(* IEC 61131-3 sources: F100R_S278_Temperville/MyController.device.xml.v3^/Plc Logic.plclogic.xml.v3^/Application.application.xml.v3^/01_Inicialização, 3 files *)

(* ---- A_Inicializacao.prg.st ---- *)
PROGRAM A_Inicializacao
VAR
	///passo para logica de inicialização do sistema
	PassoInit: INT := 0;
	ContDrive: INT := 0;
	TonInicilizacaoSistema: TON;
	xTonInicilizacaoSistemaIn: BOOL;
	xTonInicilizacaoSistemaQ: BOOL;
	TonLeituraErroInicial: TON;
	xTonLeituraErroInicialIn: BOOL;
	xTonLeituraErroInicialQ: BOOL;
	tDelayIniSystem: TON;
	tDelayIniSystemIn: BOOL;
	tDelayIniSystemQ: BOOL;
	///atraso entre os passos 0 e 1
	AtrasoPasso01: TON;
	/// tempo limite para verificar se os drives foram habilitados
	AtrasoLeituraStatus: TON;
	/// tempo de reset
	AtrasoRstErro: TON;
	delayResetaNo: TON;
	AtrasoEstabilizaRede: TON;
	/// Ativa leitura dos drives
	xAtivaLeituraErro: BOOL;
	iContadorReset: INT;
	xCanOpenOk: BOOL;
	///Flag indicativo para falha na rede CanOpen ou CanMotion
	xCanOpenFh: BOOL;
	/// Bit para habilitar drives do sistema
	xHabilitaDrives: BOOL;
	/// bit para resetar alarmes
	xRstAlarmes: BOOL;
	///------------------------------------------------------------------------//
	///Mesa Entrada
	McResetMesaEntrada: GIPLC.MC_Reset;
	McPowerMesaEntrada: GIPLC.MC_Power;
	McReadStatusMesaEntrada: GIPLC.MC_ReadStatus;
	McReadErrorMesaEntrada: GIPLC.MC_ReadAxisError;
	///Mesa Forno
	McResetMesaForno: GIPLC.MC_Reset;
	McPowerMesaForno: GIPLC.MC_Power;
	McReadStatusMesaForno: GIPLC.MC_ReadStatus;
	McReadErrorMesaForno: GIPLC.MC_ReadAxisError;
	///Mesa Resfriamento
	McResetMesaResfriador: GIPLC.MC_Reset;
	McPowerMesaResfriador: GIPLC.MC_Power;
	McReadStatusMesaResfriado: GIPLC.MC_ReadStatus;
	McReadErrorMesaResfriador: GIPLC.MC_ReadAxisError;
	///Mesa Saída
	McResetMesaSaida: GIPLC.MC_Reset;
	McPowerMesaSaida: GIPLC.MC_Power;
	McReadStatusMesaSaida: GIPLC.MC_ReadStatus;
	McReadErrorMesaSaida: GIPLC.MC_ReadAxisError;
	///Ductos Inferior 01
	McResetDutosResfriadorInf01: GIPLC.MC_Reset;
	McPowerDutosResfriadorInf01: GIPLC.MC_Power;
	McReadDutosResfriadorInf01: GIPLC.MC_ReadStatus;
	McReadErrorDutosResfriadorInf01: GIPLC.MC_ReadAxisError;
	///Ductos Superior 01
	McResetDutosResfriadorSup01: GIPLC.MC_Reset;
	McPowerDutosResfriadorSup01: GIPLC.MC_Power;
	McReadDutosResfriadorSup01: GIPLC.MC_ReadStatus;
	McReadErrorDutosResfriadorSup01: GIPLC.MC_ReadAxisError;
	///Ductos Inferior 02
	McResetDutosResfriadorInf02: GIPLC.MC_Reset;
	McPowerDutosResfriadorInf02: GIPLC.MC_Power;
	McReadDutosResfriadorInf02: GIPLC.MC_ReadStatus;
	McReadErrorDutosResfriadorInf02: GIPLC.MC_ReadAxisError;
	///Ductos Superior 02
	McResetDutosResfriadorSup02: GIPLC.MC_Reset;
	McPowerDutosResfriadorSup02: GIPLC.MC_Power;
	McReadDutosResfriadorSup02: GIPLC.MC_ReadStatus;
	McReadErrorDutosResfriadorSup02: GIPLC.MC_ReadAxisError;
	///Guilhotina01
	McResetGuilhotina01: GIPLC.MC_Reset;
	McPowerGuilhotina01: GIPLC.MC_Power;
	McReadStatusGuilhotina01: GIPLC.MC_ReadStatus;
	McReadErrorGuilhotina01: GIPLC.MC_ReadAxisError;
	///Guilhotina02
	McResetGuilhotina02: GIPLC.MC_Reset;
	McPowerGuilhotina02: GIPLC.MC_Power;
	McReadStatusGuilhotina02: GIPLC.MC_ReadStatus;
	McReadErrorGuilhotina02: GIPLC.MC_ReadAxisError;
	/// Motor Limpeza Resfriador 02
	McResetLimpResfriadorSup02: GIPLC.MC_Reset;
	McPowerLimpResfriadorSup02: GIPLC.MC_Power;
	McReadStatusLimpResfriadorSup02: GIPLC.MC_ReadStatus;
	McReadErrorLimpResfriadorSup02: GIPLC.MC_ReadAxisError;
	/// Motor Abertura Caixa do Forno
	McResetCaixaForno: GIPLC.MC_Reset;
	McPowerCaixaForno: GIPLC.MC_Power;
	McReadStatusCaixaForno: GIPLC.MC_ReadStatus;
	McReadErrorCaixaForno: GIPLC.MC_ReadAxisError;
	///Ventilador01
	McResetVentilador01: GIPLC.MC_Reset;
	McPowerVentilador01: GIPLC.MC_Power;
	McReadStatusVentilador01: GIPLC.MC_ReadStatus;
	McReadErrorVentilador01: GIPLC.MC_ReadAxisError;
	PulsoRstVent01Auto: TP;
	///Ventilador02
	McResetVentilador02: GIPLC.MC_Reset;
	McPowerVentilador02: GIPLC.MC_Power;
	McReadStatusVentilador02: GIPLC.MC_ReadStatus;
	McReadErrorVentilador02: GIPLC.MC_ReadAxisError;
	PulsoRstVent02Auto: TP;
	///Ventilador03
	McResetVentilador03: GIPLC.MC_Reset;
	McPowerVentilador03: GIPLC.MC_Power;
	McReadStatusVentilador03: GIPLC.MC_ReadStatus;
	McReadErrorVentilador03: GIPLC.MC_ReadAxisError;
	PulsoRstVent03Auto: TP;
	///Ventilador03
	McResetVentilador04: GIPLC.MC_Reset;
	McPowerVentilador04: GIPLC.MC_Power;
	McReadStatusVentilador04: GIPLC.MC_ReadStatus;
	McReadErrorVentilador04: GIPLC.MC_ReadAxisError;
	PulsoRstVent04Auto: TP;
	///Ventilador Convecção
	McResetVentConvec: GIPLC.MC_Reset;
	McPowerVentConvec: GIPLC.MC_Power;
	McReadStatusVentConvec: GIPLC.MC_ReadStatus;
	McReadErrorVentConvec: GIPLC.MC_ReadAxisError;
	///-----------------------------------------------------------------------//
	xResetErroVent03: BOOL;
	///----------------------------------------------------------------------//
	xErroDeEixo: BOOL;
	ResetaRedeCanOpen: CIA405.NMT;
	iNdevice: USINT := 1;
	testemsl: BOOL;
	AuxResetRedeCanOpen: BOOL;
	xInicializacaoOk: BOOL;
	xErroEixo: ARRAY[1..14] OF BOOL;
	xEixoHabilitado: ARRAY[1..14] OF BOOL;
	xHabilitaDriveMe: BOOL;
	xHabilitaDriveMf: BOOL;
	xHabilitaDriveMr: BOOL;
	xHabilitaDriveMs: BOOL;
	xHabilitaDriveMdI01: BOOL;
	xHabilitaDriveMdS01: BOOL;
	xHabilitaDriveMdI02: BOOL;
	xHabilitaDriveMdS02: BOOL;
	xHabilitaDriveMg01: BOOL;
	xHabilitaDriveMg02: BOOL;
	xHabilitaDriveMv01: BOOL;
	xHabilitaDriveMv02: BOOL;
	xHabilitaDriveMv03: BOOL;
	xHabilitaDriveMv04: BOOL;
	xResetErroVentilador01: BOOL;
	xResetErroVentilador02: BOOL;
	xResetErroVentilador03: BOOL;
	xResetErroVentilador04: BOOL;
	xHabilitaDriveMvC: BOOL;
	xResetErroMe: BOOL;
	xResetErroMf: BOOL;
	xResetErroMr: BOOL;
	xResetErroMs: BOOL;
	xResetErroMdS02: BOOL;
	xResetErroMg02: BOOL;
	xResetErroV03: BOOL;
	xResetErroV04: BOOL;
END_VAR

iNumResistencias:=iNumeroResistencias/2;

(* ---- ComunicacaoOpc.prg.st ---- *)
PROGRAM ComunicacaoOpc
VAR
	xEnviaSuperClp: INT;
	xRecebeClpSuper: INT;
	ton01: ton;
	ton01In: BOOL;
END_VAR
VAR_OUTPUT
	ton01Q: BOOL;
END_VAR

IF xEnviaSuperClp=1 THEN
	xEnviaSuperClp:=0;
	ton01In:=TRUE;
END_IF

ton01(IN:=ton01In , PT:=T#1000ms , Q=>ton01Q , ET=> );

IF ton01Q THEN
	xRecebeClpSuper:=1;
	ton01In:=FALSE;
END_IF

(* ---- StatusRemotasModTcpIP.prg.st ---- *)
PROGRAM StatusRemotasModTcpIP
VAR
// Variaveis Lógica StatusRemotasModTcpIP
//IOScanner Statuus
ModbusTcpIoScanner_Not_OK 	: BOOL;
ModbusTcpIoScanner_Not_Ope 	: INT;
ModbusTcpReset				: BOOL;  // Reset
//Aux HealthBits Remotas
TM3BC_ModbusTCP_1_Hb  : BOOL;
TM3BC_ModbusTCP_2_Hb  : BOOL;
TM3BC_ModbusTCP_3_Hb  : BOOL;
TM3BC_ModbusTCP_4_Hb  : BOOL;
//HealthBit Remotas not Ok
TM3BC_ModbusTCP_1_Hb_Nok  : INT;
TM3BC_ModbusTCP_2_Hb_Nok  : INT;
TM3BC_ModbusTCP_3_Hb_Nok  : INT;
TM3BC_ModbusTCP_4_Hb_Nok  : INT;
//Horários do ultimo erro
ModBusTcpAno:  ARRAY [1..10] OF UINT;
ModBusTcpMes:  ARRAY [1..10] OF UINT;
ModBusTcpDia:  ARRAY [1..10] OF UINT;
ModBusTcpHora: ARRAY [1..10] OF UINT;
ModBusTcpMin:  ARRAY [1..10] OF UINT;
ModBusTcpSeg:  ARRAY [1..10] OF UINT;

END_VAR

//Verifica IOScanner se está operacional
IF ModbusTCP_IOScanner_Gstatus = 2 THEN
	ModbusTcpIoScanner_Not_OK :=FALSE;
ELSE
	ModbusTcpIoScanner_Not_OK :=TRUE;
	ModbusTcpIoScanner_Not_Ope := ModbusTcpIoScanner_Not_Ope + 1;
	ModBusTcpAno[1]:=uAnoRealTime;
	ModBusTcpMes[1]:=uMesRealTime;
	ModBusTcpDia[1]:=uDiaRealTime;
	ModBusTcpHora[1]:=uHoraRealTime;
	ModBusTcpMin[1]:=uMinutoRealTime;
	ModBusTcpSeg[1]:=uSegundoRealTime;
END_IF

// Health bit remotas
//Verifica  remota 1 Ch0
IF ModbusTCP_IOScanner_Gstatus = 2 AND NOT TM3BC_ModbusTCP_1_Hb_Ch0 THEN
	TM3BC_ModbusTCP_1_Hb_Nok := TM3BC_ModbusTCP_1_Hb_Nok + 1;
	ModBusTcpAno[2]:=uAnoRealTime;
	ModBusTcpMes[2]:=uMesRealTime;
	ModBusTcpDia[2]:=uDiaRealTime;
	ModBusTcpHora[2]:=uHoraRealTime;
	ModBusTcpMin[2]:=uMinutoRealTime;
	ModBusTcpSeg[2]:=uSegundoRealTime;
END_IF

//Verifica remota 1 Ch1
IF ModbusTCP_IOScanner_Gstatus = 2 AND NOT TM3BC_ModbusTCP_1_Hb_Ch1 THEN
	TM3BC_ModbusTCP_1_Hb_Nok := TM3BC_ModbusTCP_1_Hb_Nok + 1;
	ModBusTcpAno[3]:=uAnoRealTime;
	ModBusTcpMes[3]:=uMesRealTime;
	ModBusTcpDia[3]:=uDiaRealTime;
	ModBusTcpHora[3]:=uHoraRealTime;
	ModBusTcpMin[3]:=uMinutoRealTime;
	ModBusTcpSeg[3]:=uSegundoRealTime;
END_IF

//Verifica remota 2 Ch2
IF ModbusTCP_IOScanner_Gstatus = 2 AND NOT TM3BC_ModbusTCP_2_Hb_Ch2 THEN
	TM3BC_ModbusTCP_2_Hb_Nok := TM3BC_ModbusTCP_2_Hb_Nok + 1;
	ModBusTcpAno[4]:=uAnoRealTime;
	ModBusTcpMes[4]:=uMesRealTime;
	ModBusTcpDia[4]:=uDiaRealTime;
	ModBusTcpHora[4]:=uHoraRealTime;
	ModBusTcpMin[4]:=uMinutoRealTime;
	ModBusTcpSeg[4]:=uSegundoRealTime;
END_IF

//Verifica remota 2 Ch3
IF ModbusTCP_IOScanner_Gstatus = 2 AND NOT TM3BC_ModbusTCP_2_Hb_Ch3 THEN
	TM3BC_ModbusTCP_2_Hb_Nok := TM3BC_ModbusTCP_2_Hb_Nok + 1;
	ModBusTcpAno[5]:=uAnoRealTime;
	ModBusTcpMes[5]:=uMesRealTime;
	ModBusTcpDia[5]:=uDiaRealTime;
	ModBusTcpHora[5]:=uHoraRealTime;
	ModBusTcpMin[5]:=uMinutoRealTime;
	ModBusTcpSeg[5]:=uSegundoRealTime;
END_IF

//Verifica remota 3 Ch4
IF ModbusTCP_IOScanner_Gstatus = 2 AND NOT TM3BC_ModbusTCP_3_Hb_Ch4 THEN
	TM3BC_ModbusTCP_3_Hb_Nok := TM3BC_ModbusTCP_3_Hb_Nok + 1;
	ModBusTcpAno[6]:=uAnoRealTime;
	ModBusTcpMes[6]:=uMesRealTime;
	ModBusTcpDia[6]:=uDiaRealTime;
	ModBusTcpHora[6]:=uHoraRealTime;
	ModBusTcpMin[6]:=uMinutoRealTime;
	ModBusTcpSeg[6]:=uSegundoRealTime;
END_IF

//Verifica remota 3 Ch5
IF ModbusTCP_IOScanner_Gstatus = 2 AND NOT TM3BC_ModbusTCP_3_Hb_Ch5 THEN
	TM3BC_ModbusTCP_3_Hb_Nok := TM3BC_ModbusTCP_3_Hb_Nok + 1;
	ModBusTcpAno[7]:=uAnoRealTime;
	ModBusTcpMes[7]:=uMesRealTime;
	ModBusTcpDia[7]:=uDiaRealTime;
	ModBusTcpHora[7]:=uHoraRealTime;
	ModBusTcpMin[7]:=uMinutoRealTime;
	ModBusTcpSeg[7]:=uSegundoRealTime;

END_IF

//Verifica remota 4 Ch6
IF ModbusTCP_IOScanner_Gstatus = 2 AND NOT TM3BC_ModbusTCP_4_Hb_Ch6 THEN
	TM3BC_ModbusTCP_4_Hb_Nok := TM3BC_ModbusTCP_4_Hb_Nok + 1;
	ModBusTcpAno[8]:=uAnoRealTime;
	ModBusTcpMes[8]:=uMesRealTime;
	ModBusTcpDia[8]:=uDiaRealTime;
	ModBusTcpHora[8]:=uHoraRealTime;
	ModBusTcpMin[8]:=uMinutoRealTime;
	ModBusTcpSeg[8]:=uSegundoRealTime;

END_IF

//Verifica remota 4 Ch7
IF ModbusTCP_IOScanner_Gstatus = 2 AND NOT TM3BC_ModbusTCP_4_Hb_Ch7 THEN
	TM3BC_ModbusTCP_4_Hb_Nok := TM3BC_ModbusTCP_4_Hb_Nok + 1;
	ModBusTcpAno[9]:=uAnoRealTime;
	ModBusTcpMes[9]:=uMesRealTime;
	ModBusTcpDia[9]:=uDiaRealTime;
	ModBusTcpHora[9]:=uHoraRealTime;
	ModBusTcpMin[9]:=uMinutoRealTime;
	ModBusTcpSeg[9]:=uSegundoRealTime;

END_IF

//Reset de contagem
IF ModbusTcpReset THEN
	ModbusTcpIoScanner_Not_OK := FALSE;
	ModbusTcpIoScanner_Not_Ope 	:= 0;
	//Aux HealthBits
	TM3BC_ModbusTCP_1_Hb  := FALSE;
	TM3BC_ModbusTCP_2_Hb  := FALSE;
	TM3BC_ModbusTCP_3_Hb  := FALSE;
	TM3BC_ModbusTCP_4_Hb  := FALSE;
	//HealthBit not Ok
	TM3BC_ModbusTCP_1_Hb_Nok  := 0;
	TM3BC_ModbusTCP_2_Hb_Nok  := 0;
	TM3BC_ModbusTCP_3_Hb_Nok  := 0;
	TM3BC_ModbusTCP_4_Hb_Nok  := 0;
	ModbusTcpReset := FALSE;
END_IF
